PROGRAM prgComEffIO
VAR
	fbCom		: FB_MqttCommunicator_V5;
	int_SSPNumber: INT;
END_VAR

fbCom(
	bConnect:= TRUE, 
	strAuthKey:= 'ENE87365342998', 
	sUserName:= , 
	sUserPassword:= , 
	eSavePositionCertificate:= eSavePositionOnPLC.ePostionHardDisk,  
	bConnected=> , 
	bError=> , 
	hrErrorCode=> , 
	eConnectionState=> , 
	eErrorMessage_Out=> );


prg_ReadDeviceName();
IF prg_ReadDeviceName.sDeviceName = '' THEN
	prg_ReadDeviceName.bStart := TRUE;
END_IF


// select user / pass according device name:

IF prg_ReadDeviceName.sDeviceName = 'EIOSM000002' THEN
	fbCom.sUserName:= '0b42849c-4998-452d-bcd9-1344b044b06a'; 
    fbCom.sUserPassword:= '8be448ae-72bb-402a-8881-f106399ccc0a';
	int_SSPNumber :=2;
ELSIF prg_ReadDeviceName.sDeviceName = 'EIOSM000003' THEN
	fbCom.sUserName:= '250c21dc-16ee-4d4b-a8b6-b80fa572657e'; 
    fbCom.sUserPassword:= '131f7038-8c5a-467b-8f48-3b98e46b3e9d';
	int_SSPNumber :=3;
ELSIF prg_ReadDeviceName.sDeviceName = 'EIOSM000004' THEN
	fbCom.sUserName:= 'c938aafa-9a8d-47b6-9d90-e88759d88525'; 
    fbCom.sUserPassword:= '03531b94-b497-4a3f-9018-b2efc52058ad';
	int_SSPNumber :=4;
ELSIF prg_ReadDeviceName.sDeviceName = 'EIOSM000001' THEN
	fbCom.sUserName:= 'c5a26c3c-d7be-49fa-bb4b-d09878f078e1'; 
    fbCom.sUserPassword:= '835df6a6-a36a-4edd-98fd-f6a495ce7360';
	int_SSPNumber :=1;
END_IF

END_PROGRAM

(* stored: Version 1.1.0.1, ProductVersion 3.1.4024.13
   POU prgComEffIO: Id {cbcd318b-bf51-484c-bcaa-d6efcdf43fe3}, SpecialFunc None *)
